DATA_BLOCK "IAI_DeviceCtl"
VAR
  IAIServo : Array[1..4] of Struct;
END_VAR
BEGIN
END_DATA_BLOCK
